(* IEC 61131-3 sources: robocpp/fuzz/corpus/pipeline, 1 file *)

(* ---- counter.st ---- *)
PROGRAM CounterDemo
VAR
    Count : INT := 0;
    Limit : INT := 3;
    Done : BOOL := FALSE;
END_VAR

IF Count < Limit THEN
    Count := Count + 1;
ELSE
    Done := TRUE;
END_IF;
END_PROGRAM
